Yaskawa INFORM job: R1-ST2-SAFE.JBI

/JOB
//NAME R1-ST2-SAFE
///FOLDERNAME FOLDER001
//POS
///NPOS 4,4,0,0,3,0
///TOOL 0
///POSTYPE PULSE
///PULSE
C00000=-3569,-156345,-136274,3722,37669,81359
C00001=-3569,-156345,-136274,3722,37669,81359
C00002=-3569,-156345,-136274,3722,37669,81359
C00003=-3569,-156344,-136273,3722,37669,81359
BC00000=85972,4,452134
BC00001=85972,4,452134
BC00002=85972,4,452134
BC00003=85972,837360,452132
///POSTYPE BASE
///RECTAN
///RCONF 0,0,0,0,0,0,0,0,0,0,0,0,0,0,0,0,0,0,0,0,0,0,0,0
BP00001=720.111,37.947,1642.122
BP00002=1602.617,32.863,1148.397
///POSTYPE ROBOT
BP00003=1488.326,670.297,1439.201
//INST
///DATE 2023/07/10 16:57
///ATTR SC,RW
///GROUP1 RB1,BS1
NOP
SFTOF
REFP 1 C00000 BC00000
GETS PX001 $PX011
CNVRT PX001 PX001 RF
GETS PX002 $PX001
CNVRT PX002 PX002 RF
SUB BP002 BP001
SET BP003 BP002
SFTON BP003
MOVJ C00001 BC00001 VJ=50.00
SFTOF
SETE BP003 (1) 0
SETE BP003 (3) 0
SFTON BP003
MOVJ C00002 BC00002 VJ=25.00
SFTOF
MOVJ C00003 BC00003 VJ=25.00
END
